PROGRAM MAIN
VAR
	fbGen : GEN;
	nOut: INT;
END_VAR

fbGen(
	MODE:= SINE, 
	BASE:= TRUE, 
	PERIOD:= T#200MS, 
	CYCLES:= 200, 
	AMPLITUDE:= 10, 
	RESET:= , 
	OUT=> nOut);

END_PROGRAM

(* stored: Version 1.1.0.1, ProductVersion 3.1.4024.12
   POU MAIN: Id {a27a9b3e-2c42-4f26-a437-74b050783276}, SpecialFunc None *)
